FUNCTION_BLOCK PUBLIC SINT_TO_TestSuite EXTENDS TcUnit.FB_TestSuite
VAR
END_VAR

Check_SINT_TO_BOOL_Max();
Check_SINT_TO_BOOL_Min();
Check_SINT_TO_BYTE_Max();
Check_SINT_TO_BYTE_Min();
Check_SINT_TO_BYTE_TooLow();
Check_SINT_TO_WORD_Max();
Check_SINT_TO_WORD_Min();
Check_SINT_TO_WORD_TooLow();
Check_SINT_TO_DWORD_Max();
Check_SINT_TO_DWORD_Min();
Check_SINT_TO_DWORD_TooLow();
Check_SINT_TO_LWORD_Max();
Check_SINT_TO_LWORD_Min();
Check_SINT_TO_LWORD_TooLow();
Check_SINT_TO_SINT_Max();
Check_SINT_TO_SINT_Min();
Check_SINT_TO_INT_Max();
Check_SINT_TO_INT_Min();
Check_SINT_TO_DINT_Max();
Check_SINT_TO_DINT_Min();
Check_SINT_TO_LINT_Max();
Check_SINT_TO_LINT_Min();
Check_SINT_TO_USINT_Max();
Check_SINT_TO_USINT_Min();
Check_SINT_TO_USINT_TooLow();
Check_SINT_TO_UINT_Max();
Check_SINT_TO_UINT_Min();
Check_SINT_TO_UINT_TooLow();
Check_SINT_TO_UDINT_Max();
Check_SINT_TO_UDINT_Min();
Check_SINT_TO_UDINT_TooLow();
Check_SINT_TO_ULINT_Max();
Check_SINT_TO_ULINT_Min();
Check_SINT_TO_ULINT_TooLow();
Check_SINT_TO_REAL_Max();
Check_SINT_TO_REAL_Min();
Check_SINT_TO_LREAL_Max();
Check_SINT_TO_LREAL_Min();
Check_SINT_TO_TIME_Max();
Check_SINT_TO_TIME_Min();
Check_SINT_TO_TIME_TooLow();
Check_SINT_TO_TOD_Max();
Check_SINT_TO_TOD_Min();
Check_SINT_TO_TOD_TooLow();
Check_SINT_TO_DATE_Max();
Check_SINT_TO_DATE_Min();
Check_SINT_TO_DATE_TooLow();
Check_SINT_TO_DT_Max();
Check_SINT_TO_DT_Min();
Check_SINT_TO_DT_TooLow();
Check_SINT_TO_STRING_Max();
Check_SINT_TO_STRING_Min();

METHOD PUBLIC Check_SINT_TO_BOOL_Min
VAR
	value : SINT := DatatypeLimits.SINT_MIN_VALUE;
	actual : BOOL;
	converted : BOOL;
	equal : BOOL;
END_VAR
TEST('Check_SINT_TO_BOOL_Min');

// @TEST-RUN
converted := TryConvert_SINT_TO_Destination(value, actual);
equal := actual = SINT_TO_BOOL(value);

// @TEST-ASSERT
AssertTrue(Condition := equal, Message := 'Did not convert SINT to BOOL correctly');
AssertTrue(Condition := converted, Message := 'Did not report SINT to BOOL conversion was successful');

TEST_FINISHED();
END_METHOD

METHOD PUBLIC Check_SINT_TO_BOOL_Max
VAR
	value : SINT := DatatypeLimits.SINT_MAX_VALUE;
	actual : BOOL;
	converted : BOOL;
	equal : BOOL;
END_VAR
TEST('Check_SINT_TO_BOOL_Max');

// @TEST-RUN
converted := TryConvert_SINT_TO_Destination(value, actual);
equal := actual = SINT_TO_BOOL(value);

// @TEST-ASSERT
AssertTrue(Condition := equal, Message := 'Did not convert SINT to BOOL correctly');
AssertTrue(Condition := converted, Message := 'Did not report SINT to BOOL conversion was successful');

TEST_FINISHED();
END_METHOD

METHOD PUBLIC Check_SINT_TO_BYTE_Min
VAR
	value : SINT := DatatypeLimits.MIN_VALUE_OF_SINT_WHICH_CAN_BE_HELD_IN_A_BYTE;
	actual : BYTE;
	converted : BOOL;
	equal : BOOL;
END_VAR
TEST('Check_SINT_TO_BYTE_Min');

// @TEST-RUN
converted := TryConvert_SINT_TO_Destination(value, actual);
equal := actual = SINT_TO_BYTE(value);

// @TEST-ASSERT
AssertTrue(Condition := equal, Message := 'Did not convert SINT to BYTE correctly');
AssertTrue(Condition := converted, Message := 'Did not report SINT to BYTE conversion was successful');

TEST_FINISHED();
END_METHOD

METHOD PUBLIC Check_SINT_TO_BYTE_TooLow
VAR
	value : SINT := DatatypeLimits.SINT_MIN_VALUE;
	actual : BYTE;
	converted : BOOL;
END_VAR
TEST('Check_SINT_TO_BYTE_TooLow');

// @TEST-RUN
converted := TryConvert_SINT_TO_Destination(value, actual);

// @TEST-ASSERT
AssertFalse(Condition := converted, Message := 'Did not report SINT to BYTE conversion was prevented');

TEST_FINISHED();
END_METHOD

METHOD PUBLIC Check_SINT_TO_BYTE_Max
VAR
	value : SINT := DatatypeLimits.SINT_MAX_VALUE;
	actual : BYTE;
	converted : BOOL;
	equal : BOOL;
END_VAR
TEST('Check_SINT_TO_BYTE_Max');

// @TEST-RUN
converted := TryConvert_SINT_TO_Destination(value, actual);
equal := actual = SINT_TO_BYTE(value);

// @TEST-ASSERT
AssertTrue(Condition := equal, Message := 'Did not convert SINT to BYTE correctly');
AssertTrue(Condition := converted, Message := 'Did not report SINT to BYTE conversion was successful');

TEST_FINISHED();
END_METHOD

METHOD PUBLIC Check_SINT_TO_DATE_Min
VAR
	value : SINT := DatatypeLimits.MIN_VALUE_OF_SINT_WHICH_CAN_BE_HELD_IN_A_DATE;
	actual : DATE;
	converted : BOOL;
	equal : BOOL;
END_VAR
TEST('Check_SINT_TO_DATE_Min');

// @TEST-RUN
converted := TryConvert_SINT_TO_Destination(value, actual);
equal := actual = SINT_TO_DATE(value);

// @TEST-ASSERT
AssertTrue(Condition := equal, Message := 'Did not convert SINT to DATE correctly');
AssertTrue(Condition := converted, Message := 'Did not report SINT to DATE conversion was successful');

TEST_FINISHED();
END_METHOD

METHOD PUBLIC Check_SINT_TO_DATE_TooLow
VAR
	value : SINT := DatatypeLimits.SINT_MIN_VALUE;
	actual : DATE;
	converted : BOOL;
END_VAR
TEST('Check_SINT_TO_DATE_TooLow');

// @TEST-RUN
converted := TryConvert_SINT_TO_Destination(value, actual);

// @TEST-ASSERT
AssertFalse(Condition := converted, Message := 'Did not report SINT to DATE conversion was prevented');

TEST_FINISHED();
END_METHOD

METHOD PUBLIC Check_SINT_TO_DATE_Max
VAR
	value : SINT := DatatypeLimits.SINT_MAX_VALUE;
	actual : DATE;
	converted : BOOL;
	equal : BOOL;
END_VAR
TEST('Check_SINT_TO_DATE_Max');

// @TEST-RUN
converted := TryConvert_SINT_TO_Destination(value, actual);
equal := actual = SINT_TO_DATE(value);

// @TEST-ASSERT
AssertTrue(Condition := equal, Message := 'Did not convert SINT to DATE correctly');
AssertTrue(Condition := converted, Message := 'Did not report SINT to DATE conversion was successful');

TEST_FINISHED();
END_METHOD

METHOD PUBLIC Check_SINT_TO_DINT_Min
VAR
	value : SINT := DatatypeLimits.SINT_MIN_VALUE;
	actual : DINT;
	converted : BOOL;
	equal : BOOL;
END_VAR
TEST('Check_SINT_TO_DINT_Min');

// @TEST-RUN
converted := TryConvert_SINT_TO_Destination(value, actual);
equal := actual = SINT_TO_DINT(value);

// @TEST-ASSERT
AssertTrue(Condition := equal, Message := 'Did not convert SINT to DINT correctly');
AssertTrue(Condition := converted, Message := 'Did not report SINT to DINT conversion was successful');

TEST_FINISHED();
END_METHOD

METHOD PUBLIC Check_SINT_TO_DINT_Max
VAR
	value : SINT := DatatypeLimits.SINT_MAX_VALUE;
	actual : DINT;
	converted : BOOL;
	equal : BOOL;
END_VAR
TEST('Check_SINT_TO_DINT_Max');

// @TEST-RUN
converted := TryConvert_SINT_TO_Destination(value, actual);
equal := actual = SINT_TO_DINT(value);

// @TEST-ASSERT
AssertTrue(Condition := equal, Message := 'Did not convert SINT to DINT correctly');
AssertTrue(Condition := converted, Message := 'Did not report SINT to DINT conversion was successful');

TEST_FINISHED();
END_METHOD

METHOD PUBLIC Check_SINT_TO_DT_Min
VAR
	value : SINT := DatatypeLimits.MIN_VALUE_OF_SINT_WHICH_CAN_BE_HELD_IN_A_DT;
	actual : DT;
	converted : BOOL;
	equal : BOOL;
END_VAR
TEST('Check_SINT_TO_DT_Min');

// @TEST-RUN
converted := TryConvert_SINT_TO_Destination(value, actual);
equal := actual = SINT_TO_DT(value);

// @TEST-ASSERT
AssertTrue(Condition := equal, Message := 'Did not convert SINT to DT correctly');
AssertTrue(Condition := converted, Message := 'Did not report SINT to DT conversion was successful');

TEST_FINISHED();
END_METHOD

METHOD PUBLIC Check_SINT_TO_DT_TooLow
VAR
	value : SINT := DatatypeLimits.SINT_MIN_VALUE;
	actual : DT;
	converted : BOOL;
END_VAR
TEST('Check_SINT_TO_DT_TooLow');

// @TEST-RUN
converted := TryConvert_SINT_TO_Destination(value, actual);

// @TEST-ASSERT
AssertFalse(Condition := converted, Message := 'Did not report SINT to DT conversion was prevented');

TEST_FINISHED();
END_METHOD

METHOD PUBLIC Check_SINT_TO_DT_Max
VAR
	value : SINT := DatatypeLimits.SINT_MAX_VALUE;
	actual : DT;
	converted : BOOL;
	equal : BOOL;
END_VAR
TEST('Check_SINT_TO_DT_Max');

// @TEST-RUN
converted := TryConvert_SINT_TO_Destination(value, actual);
equal := actual = SINT_TO_DT(value);

// @TEST-ASSERT
AssertTrue(Condition := equal, Message := 'Did not convert SINT to DT correctly');
AssertTrue(Condition := converted, Message := 'Did not report SINT to DT conversion was successful');

TEST_FINISHED();
END_METHOD

METHOD PUBLIC Check_SINT_TO_DWORD_Min
VAR
	value : SINT := DatatypeLimits.MIN_VALUE_OF_SINT_WHICH_CAN_BE_HELD_IN_A_DWORD;
	actual : DWORD;
	converted : BOOL;
	equal : BOOL;
END_VAR
TEST('Check_SINT_TO_DWORD_Min');

// @TEST-RUN
converted := TryConvert_SINT_TO_Destination(value, actual);
equal := actual = SINT_TO_DWORD(value);

// @TEST-ASSERT
AssertTrue(Condition := equal, Message := 'Did not convert SINT to DWORD correctly');
AssertTrue(Condition := converted, Message := 'Did not report SINT to DWORD conversion was successful');

TEST_FINISHED();
END_METHOD

METHOD PUBLIC Check_SINT_TO_DWORD_TooLow
VAR
	value : SINT := DatatypeLimits.SINT_MIN_VALUE;
	actual : DWORD;
	converted : BOOL;
END_VAR
TEST('Check_SINT_TO_DWORD_TooLow');

// @TEST-RUN
converted := TryConvert_SINT_TO_Destination(value, actual);

// @TEST-ASSERT
AssertFalse(Condition := converted, Message := 'Did not report SINT to DWORD conversion was prevented');

TEST_FINISHED();
END_METHOD

METHOD PUBLIC Check_SINT_TO_DWORD_Max
VAR
	value : SINT := DatatypeLimits.SINT_MAX_VALUE;
	actual : DWORD;
	converted : BOOL;
	equal : BOOL;
END_VAR
TEST('Check_SINT_TO_DWORD_Max');

// @TEST-RUN
converted := TryConvert_SINT_TO_Destination(value, actual);
equal := actual = SINT_TO_DWORD(value);

// @TEST-ASSERT
AssertTrue(Condition := equal, Message := 'Did not convert SINT to DWORD correctly');
AssertTrue(Condition := converted, Message := 'Did not report SINT to DWORD conversion was successful');

TEST_FINISHED();
END_METHOD

METHOD PUBLIC Check_SINT_TO_INT_Min
VAR
	value : SINT := DatatypeLimits.SINT_MIN_VALUE;
	actual : INT;
	converted : BOOL;
	equal : BOOL;
END_VAR
TEST('Check_SINT_TO_INT_Min');

// @TEST-RUN
converted := TryConvert_SINT_TO_Destination(value, actual);
equal := actual = SINT_TO_INT(value);

// @TEST-ASSERT
AssertTrue(Condition := equal, Message := 'Did not convert SINT to INT correctly');
AssertTrue(Condition := converted, Message := 'Did not report SINT to INT conversion was successful');

TEST_FINISHED();
END_METHOD

METHOD PUBLIC Check_SINT_TO_INT_Max
VAR
	value : SINT := DatatypeLimits.SINT_MAX_VALUE;
	actual : INT;
	converted : BOOL;
	equal : BOOL;
END_VAR
TEST('Check_SINT_TO_INT_Max');

// @TEST-RUN
converted := TryConvert_SINT_TO_Destination(value, actual);
equal := actual = SINT_TO_INT(value);

// @TEST-ASSERT
AssertTrue(Condition := equal, Message := 'Did not convert SINT to INT correctly');
AssertTrue(Condition := converted, Message := 'Did not report SINT to INT conversion was successful');

TEST_FINISHED();
END_METHOD

METHOD PUBLIC Check_SINT_TO_LINT_Min
VAR
	value : SINT := DatatypeLimits.SINT_MIN_VALUE;
	actual : LINT;
	converted : BOOL;
	equal : BOOL;
END_VAR
TEST('Check_SINT_TO_LINT_Min');

// @TEST-RUN
converted := TryConvert_SINT_TO_Destination(value, actual);
equal := actual = SINT_TO_LINT(value);

// @TEST-ASSERT
AssertTrue(Condition := equal, Message := 'Did not convert SINT to LINT correctly');
AssertTrue(Condition := converted, Message := 'Did not report SINT to LINT conversion was successful');

TEST_FINISHED();
END_METHOD

METHOD PUBLIC Check_SINT_TO_LINT_Max
VAR
	value : SINT := DatatypeLimits.SINT_MAX_VALUE;
	actual : LINT;
	converted : BOOL;
	equal : BOOL;
END_VAR
TEST('Check_SINT_TO_LINT_Max');

// @TEST-RUN
converted := TryConvert_SINT_TO_Destination(value, actual);
equal := actual = SINT_TO_LINT(value);

// @TEST-ASSERT
AssertTrue(Condition := equal, Message := 'Did not convert SINT to LINT correctly');
AssertTrue(Condition := converted, Message := 'Did not report SINT to LINT conversion was successful');

TEST_FINISHED();
END_METHOD

METHOD PUBLIC Check_SINT_TO_LREAL_Min
VAR
	value : SINT := DatatypeLimits.SINT_MIN_VALUE;
	actual : LREAL;
	converted : BOOL;
	equal : BOOL;
END_VAR
TEST('Check_SINT_TO_LREAL_Min');

// @TEST-RUN
converted := TryConvert_SINT_TO_Destination(value, actual);
equal := actual = SINT_TO_LREAL(value);

// @TEST-ASSERT
AssertTrue(Condition := equal, Message := 'Did not convert SINT to LREAL correctly');
AssertTrue(Condition := converted, Message := 'Did not report SINT to LREAL conversion was successful');

TEST_FINISHED();
END_METHOD

METHOD PUBLIC Check_SINT_TO_LREAL_Max
VAR
	value : SINT := DatatypeLimits.SINT_MAX_VALUE;
	actual : LREAL;
	converted : BOOL;
	equal : BOOL;
END_VAR
TEST('Check_SINT_TO_LREAL_Max');

// @TEST-RUN
converted := TryConvert_SINT_TO_Destination(value, actual);
equal := actual = SINT_TO_LREAL(value);

// @TEST-ASSERT
AssertTrue(Condition := equal, Message := 'Did not convert SINT to LREAL correctly');
AssertTrue(Condition := converted, Message := 'Did not report SINT to LREAL conversion was successful');

TEST_FINISHED();
END_METHOD

METHOD PUBLIC Check_SINT_TO_LWORD_Min
VAR
	value : SINT := DatatypeLimits.MIN_VALUE_OF_SINT_WHICH_CAN_BE_HELD_IN_A_LWORD;
	actual : LWORD;
	converted : BOOL;
	equal : BOOL;
END_VAR
TEST('Check_SINT_TO_LWORD_Min');

// @TEST-RUN
converted := TryConvert_SINT_TO_Destination(value, actual);
equal := actual = SINT_TO_LWORD(value);

// @TEST-ASSERT
AssertTrue(Condition := equal, Message := 'Did not convert SINT to LWORD correctly');
AssertTrue(Condition := converted, Message := 'Did not report SINT to LWORD conversion was successful');

TEST_FINISHED();
END_METHOD

METHOD PUBLIC Check_SINT_TO_LWORD_TooLow
VAR
	value : SINT := DatatypeLimits.SINT_MIN_VALUE;
	actual : LWORD;
	converted : BOOL;
END_VAR
TEST('Check_SINT_TO_LWORD_TooLow');

// @TEST-RUN
converted := TryConvert_SINT_TO_Destination(value, actual);

// @TEST-ASSERT
AssertFalse(Condition := converted, Message := 'Did not report SINT to LWORD conversion was prevented');

TEST_FINISHED();
END_METHOD

METHOD PUBLIC Check_SINT_TO_LWORD_Max
VAR
	value : SINT := DatatypeLimits.SINT_MAX_VALUE;
	actual : LWORD;
	converted : BOOL;
	equal : BOOL;
END_VAR
TEST('Check_SINT_TO_LWORD_Max');

// @TEST-RUN
converted := TryConvert_SINT_TO_Destination(value, actual);
equal := actual = SINT_TO_LWORD(value);

// @TEST-ASSERT
AssertTrue(Condition := equal, Message := 'Did not convert SINT to LWORD correctly');
AssertTrue(Condition := converted, Message := 'Did not report SINT to LWORD conversion was successful');

TEST_FINISHED();
END_METHOD

METHOD PUBLIC Check_SINT_TO_REAL_Min
VAR
	value : SINT := DatatypeLimits.SINT_MIN_VALUE;
	actual : REAL;
	converted : BOOL;
	equal : BOOL;
END_VAR
TEST('Check_SINT_TO_REAL_Min');

// @TEST-RUN
converted := TryConvert_SINT_TO_Destination(value, actual);
equal := actual = SINT_TO_REAL(value);

// @TEST-ASSERT
AssertTrue(Condition := equal, Message := 'Did not convert SINT to REAL correctly');
AssertTrue(Condition := converted, Message := 'Did not report SINT to REAL conversion was successful');

TEST_FINISHED();
END_METHOD

METHOD PUBLIC Check_SINT_TO_REAL_Max
VAR
	value : SINT := DatatypeLimits.SINT_MAX_VALUE;
	actual : REAL;
	converted : BOOL;
	equal : BOOL;
END_VAR
TEST('Check_SINT_TO_REAL_Max');

// @TEST-RUN
converted := TryConvert_SINT_TO_Destination(value, actual);
equal := actual = SINT_TO_REAL(value);

// @TEST-ASSERT
AssertTrue(Condition := equal, Message := 'Did not convert SINT to REAL correctly');
AssertTrue(Condition := converted, Message := 'Did not report SINT to REAL conversion was successful');

TEST_FINISHED();
END_METHOD

METHOD PUBLIC Check_SINT_TO_SINT_Min
VAR
	value : SINT := DatatypeLimits.SINT_MIN_VALUE;
	actual : SINT;
	converted : BOOL;
	equal : BOOL;
END_VAR
TEST('Check_SINT_TO_SINT_Min');

// @TEST-RUN
converted := TryConvert_SINT_TO_Destination(value, actual);
equal := actual = value;

// @TEST-ASSERT
AssertTrue(Condition := equal, Message := 'Did not convert SINT to SINT correctly');
AssertTrue(Condition := converted, Message := 'Did not report SINT to SINT conversion was successful');

TEST_FINISHED();
END_METHOD

METHOD PUBLIC Check_SINT_TO_SINT_Max
VAR
	value : SINT := DatatypeLimits.SINT_MAX_VALUE;
	actual : SINT;
	converted : BOOL;
	equal : BOOL;
END_VAR
TEST('Check_SINT_TO_SINT_Max');

// @TEST-RUN
converted := TryConvert_SINT_TO_Destination(value, actual);
equal := actual = value;

// @TEST-ASSERT
AssertTrue(Condition := equal, Message := 'Did not convert SINT to SINT correctly');
AssertTrue(Condition := converted, Message := 'Did not report SINT to SINT conversion was successful');

TEST_FINISHED();
END_METHOD

METHOD PUBLIC Check_SINT_TO_STRING_Min
VAR
	value : SINT := DatatypeLimits.SINT_MIN_VALUE;
	actual : STRING;
	converted : BOOL;
	equal : BOOL;
END_VAR
TEST('Check_SINT_TO_STRING_Min');

// @TEST-RUN
converted := TryConvert_SINT_TO_Destination(value, actual);
equal := actual = SINT_TO_STRING(value);

// @TEST-ASSERT
AssertTrue(Condition := equal, Message := 'Did not convert SINT to STRING correctly');
AssertTrue(Condition := converted, Message := 'Did not report SINT to STRING conversion was successful');

TEST_FINISHED();
END_METHOD

METHOD PUBLIC Check_SINT_TO_STRING_Max
VAR
	value : SINT := DatatypeLimits.SINT_MAX_VALUE;
	actual : STRING;
	converted : BOOL;
	equal : BOOL;
END_VAR
TEST('Check_SINT_TO_STRING_Max');

// @TEST-RUN
converted := TryConvert_SINT_TO_Destination(value, actual);
equal := actual = SINT_TO_STRING(value);

// @TEST-ASSERT
AssertTrue(Condition := equal, Message := 'Did not convert SINT to STRING correctly');
AssertTrue(Condition := converted, Message := 'Did not report SINT to STRING conversion was successful');

TEST_FINISHED();
END_METHOD

METHOD PUBLIC Check_SINT_TO_TIME_Min
VAR
	value : SINT := DatatypeLimits.MIN_VALUE_OF_SINT_WHICH_CAN_BE_HELD_IN_A_TIME;
	actual : TIME;
	converted : BOOL;
	equal : BOOL;
END_VAR
TEST('Check_SINT_TO_TIME_Min');

// @TEST-RUN
converted := TryConvert_SINT_TO_Destination(value, actual);
equal := actual = SINT_TO_TIME(value);

// @TEST-ASSERT
AssertTrue(Condition := equal, Message := 'Did not convert SINT to TIME correctly');
AssertTrue(Condition := converted, Message := 'Did not report SINT to TIME conversion was successful');

TEST_FINISHED();
END_METHOD

METHOD PUBLIC Check_SINT_TO_TIME_TooLow
VAR
	value : SINT := DatatypeLimits.SINT_MIN_VALUE;
	actual : TIME;
	converted : BOOL;
END_VAR
TEST('Check_SINT_TO_TIME_TooLow');

// @TEST-RUN
converted := TryConvert_SINT_TO_Destination(value, actual);

// @TEST-ASSERT
AssertFalse(Condition := converted, Message := 'Did not report SINT to TIME conversion was prevented');

TEST_FINISHED();
END_METHOD

METHOD PUBLIC Check_SINT_TO_TIME_Max
VAR
	value : SINT := DatatypeLimits.SINT_MAX_VALUE;
	actual : TIME;
	converted : BOOL;
	equal : BOOL;
END_VAR
TEST('Check_SINT_TO_TIME_Max');

// @TEST-RUN
converted := TryConvert_SINT_TO_Destination(value, actual);
equal := actual = SINT_TO_TIME(value);

// @TEST-ASSERT
AssertTrue(Condition := equal, Message := 'Did not convert SINT to TIME correctly');
AssertTrue(Condition := converted, Message := 'Did not report SINT to TIME conversion was successful');

TEST_FINISHED();
END_METHOD

METHOD PUBLIC Check_SINT_TO_TOD_Min
VAR
	value : SINT := DatatypeLimits.MIN_VALUE_OF_SINT_WHICH_CAN_BE_HELD_IN_A_TOD;
	actual : TOD;
	converted : BOOL;
	equal : BOOL;
END_VAR
TEST('Check_SINT_TO_TOD_Min');

// @TEST-RUN
converted := TryConvert_SINT_TO_Destination(value, actual);
equal := actual = SINT_TO_TOD(value);

// @TEST-ASSERT
AssertTrue(Condition := equal, Message := 'Did not convert SINT to TOD correctly');
AssertTrue(Condition := converted, Message := 'Did not report SINT to TOD conversion was successful');

TEST_FINISHED();
END_METHOD

METHOD PUBLIC Check_SINT_TO_TOD_TooLow
VAR
	value : SINT := DatatypeLimits.SINT_MIN_VALUE;
	actual : TOD;
	converted : BOOL;
END_VAR
TEST('Check_SINT_TO_TOD_TooLow');

// @TEST-RUN
converted := TryConvert_SINT_TO_Destination(value, actual);

// @TEST-ASSERT
AssertFalse(Condition := converted, Message := 'Did not report SINT to TOD conversion was prevented');

TEST_FINISHED();
END_METHOD

METHOD PUBLIC Check_SINT_TO_TOD_Max
VAR
	value : SINT := DatatypeLimits.SINT_MAX_VALUE;
	actual : TOD;
	converted : BOOL;
	equal : BOOL;
END_VAR
TEST('Check_SINT_TO_TOD_Max');

// @TEST-RUN
converted := TryConvert_SINT_TO_Destination(value, actual);
equal := actual = SINT_TO_TOD(value);

// @TEST-ASSERT
AssertTrue(Condition := equal, Message := 'Did not convert SINT to TOD correctly');
AssertTrue(Condition := converted, Message := 'Did not report SINT to TOD conversion was successful');

TEST_FINISHED();
END_METHOD

METHOD PUBLIC Check_SINT_TO_UDINT_Min
VAR
	value : SINT := DatatypeLimits.MIN_VALUE_OF_SINT_WHICH_CAN_BE_HELD_IN_A_UDINT;
	actual : UDINT;
	converted : BOOL;
	equal : BOOL;
END_VAR
TEST('Check_SINT_TO_UDINT_Min');

// @TEST-RUN
converted := TryConvert_SINT_TO_Destination(value, actual);
equal := actual = SINT_TO_UDINT(value);

// @TEST-ASSERT
AssertTrue(Condition := equal, Message := 'Did not convert SINT to UDINT correctly');
AssertTrue(Condition := converted, Message := 'Did not report SINT to UDINT conversion was successful');

TEST_FINISHED();
END_METHOD

METHOD PUBLIC Check_SINT_TO_UDINT_TooLow
VAR
	value : SINT := DatatypeLimits.SINT_MIN_VALUE;
	actual : UDINT;
	converted : BOOL;
END_VAR
TEST('Check_SINT_TO_UDINT_TooLow');

// @TEST-RUN
converted := TryConvert_SINT_TO_Destination(value, actual);

// @TEST-ASSERT
AssertFalse(Condition := converted, Message := 'Did not report SINT to UDINT conversion was prevented');

TEST_FINISHED();
END_METHOD

METHOD PUBLIC Check_SINT_TO_UDINT_Max
VAR
	value : SINT := DatatypeLimits.SINT_MAX_VALUE;
	actual : UDINT;
	converted : BOOL;
	equal : BOOL;
END_VAR
TEST('Check_SINT_TO_UDINT_Max');

// @TEST-RUN
converted := TryConvert_SINT_TO_Destination(value, actual);
equal := actual = SINT_TO_UDINT(value);

// @TEST-ASSERT
AssertTrue(Condition := equal, Message := 'Did not convert SINT to UDINT correctly');
AssertTrue(Condition := converted, Message := 'Did not report SINT to UDINT conversion was successful');

TEST_FINISHED();
END_METHOD

METHOD PUBLIC Check_SINT_TO_UINT_Min
VAR
	value : SINT := DatatypeLimits.MIN_VALUE_OF_SINT_WHICH_CAN_BE_HELD_IN_A_UINT;
	actual : UINT;
	converted : BOOL;
	equal : BOOL;
END_VAR
TEST('Check_SINT_TO_UINT_Min');

// @TEST-RUN
converted := TryConvert_SINT_TO_Destination(value, actual);
equal := actual = SINT_TO_UINT(value);

// @TEST-ASSERT
AssertTrue(Condition := equal, Message := 'Did not convert SINT to UINT correctly');
AssertTrue(Condition := converted, Message := 'Did not report SINT to UINT conversion was successful');

TEST_FINISHED();
END_METHOD

METHOD PUBLIC Check_SINT_TO_UINT_TooLow
VAR
	value : SINT := DatatypeLimits.SINT_MIN_VALUE;
	actual : UINT;
	converted : BOOL;
END_VAR
TEST('Check_SINT_TO_UINT_TooLow');

// @TEST-RUN
converted := TryConvert_SINT_TO_Destination(value, actual);

// @TEST-ASSERT
AssertFalse(Condition := converted, Message := 'Did not report SINT to UINT conversion was prevented');

TEST_FINISHED();
END_METHOD

METHOD PUBLIC Check_SINT_TO_UINT_Max
VAR
	value : SINT := DatatypeLimits.SINT_MAX_VALUE;
	actual : UINT;
	converted : BOOL;
	equal : BOOL;
END_VAR
TEST('Check_SINT_TO_UINT_Max');

// @TEST-RUN
converted := TryConvert_SINT_TO_Destination(value, actual);
equal := actual = SINT_TO_UINT(value);

// @TEST-ASSERT
AssertTrue(Condition := equal, Message := 'Did not convert SINT to UINT correctly');
AssertTrue(Condition := converted, Message := 'Did not report SINT to UINT conversion was successful');

TEST_FINISHED();
END_METHOD

METHOD PUBLIC Check_SINT_TO_ULINT_Min
VAR
	value : SINT := DatatypeLimits.MIN_VALUE_OF_SINT_WHICH_CAN_BE_HELD_IN_A_ULINT;
	actual : ULINT;
	converted : BOOL;
	equal : BOOL;
END_VAR
TEST('Check_SINT_TO_ULINT_Min');

// @TEST-RUN
converted := TryConvert_SINT_TO_Destination(value, actual);
equal := actual = SINT_TO_ULINT(value);

// @TEST-ASSERT
AssertTrue(Condition := equal, Message := 'Did not convert SINT to ULINT correctly');
AssertTrue(Condition := converted, Message := 'Did not report SINT to ULINT conversion was successful');

TEST_FINISHED();
END_METHOD

METHOD PUBLIC Check_SINT_TO_ULINT_TooLow
VAR
	value : SINT := DatatypeLimits.SINT_MIN_VALUE;
	actual : ULINT;
	converted : BOOL;
END_VAR
TEST('Check_SINT_TO_ULINT_TooLow');

// @TEST-RUN
converted := TryConvert_SINT_TO_Destination(value, actual);

// @TEST-ASSERT
AssertFalse(Condition := converted, Message := 'Did not report SINT to ULINT conversion was prevented');

TEST_FINISHED();
END_METHOD

METHOD PUBLIC Check_SINT_TO_ULINT_Max
VAR
	value : SINT := DatatypeLimits.SINT_MAX_VALUE;
	actual : ULINT;
	converted : BOOL;
	equal : BOOL;
END_VAR
TEST('Check_SINT_TO_ULINT_Max');

// @TEST-RUN
converted := TryConvert_SINT_TO_Destination(value, actual);
equal := actual = SINT_TO_ULINT(value);

// @TEST-ASSERT
AssertTrue(Condition := equal, Message := 'Did not convert SINT to ULINT correctly');
AssertTrue(Condition := converted, Message := 'Did not report SINT to ULINT conversion was successful');

TEST_FINISHED();
END_METHOD

METHOD PUBLIC Check_SINT_TO_USINT_Min
VAR
	value : SINT := DatatypeLimits.MIN_VALUE_OF_SINT_WHICH_CAN_BE_HELD_IN_A_USINT;
	actual : USINT;
	converted : BOOL;
	equal : BOOL;
END_VAR
TEST('Check_SINT_TO_USINT_Min');

// @TEST-RUN
converted := TryConvert_SINT_TO_Destination(value, actual);
equal := actual = SINT_TO_USINT(value);

// @TEST-ASSERT
AssertTrue(Condition := equal, Message := 'Did not convert SINT to USINT correctly');
AssertTrue(Condition := converted, Message := 'Did not report SINT to USINT conversion was successful');

TEST_FINISHED();
END_METHOD

METHOD PUBLIC Check_SINT_TO_USINT_TooLow
VAR
	value : SINT := DatatypeLimits.SINT_MIN_VALUE;
	actual : USINT;
	converted : BOOL;
END_VAR
TEST('Check_SINT_TO_USINT_TooLow');

// @TEST-RUN
converted := TryConvert_SINT_TO_Destination(value, actual);

// @TEST-ASSERT
AssertFalse(Condition := converted, Message := 'Did not report SINT to USINT conversion was prevented');

TEST_FINISHED();
END_METHOD

METHOD PUBLIC Check_SINT_TO_USINT_Max
VAR
	value : SINT := DatatypeLimits.SINT_MAX_VALUE;
	actual : USINT;
	converted : BOOL;
	equal : BOOL;
END_VAR
TEST('Check_SINT_TO_USINT_Max');

// @TEST-RUN
converted := TryConvert_SINT_TO_Destination(value, actual);
equal := actual = SINT_TO_USINT(value);

// @TEST-ASSERT
AssertTrue(Condition := equal, Message := 'Did not convert SINT to USINT correctly');
AssertTrue(Condition := converted, Message := 'Did not report SINT to USINT conversion was successful');

TEST_FINISHED();
END_METHOD

METHOD PUBLIC Check_SINT_TO_WORD_Min
VAR
	value : SINT := DatatypeLimits.MIN_VALUE_OF_SINT_WHICH_CAN_BE_HELD_IN_A_WORD;
	actual : WORD;
	converted : BOOL;
	equal : BOOL;
END_VAR
TEST('Check_SINT_TO_WORD_Min');

// @TEST-RUN
converted := TryConvert_SINT_TO_Destination(value, actual);
equal := actual = SINT_TO_WORD(value);

// @TEST-ASSERT
AssertTrue(Condition := equal, Message := 'Did not convert SINT to WORD correctly');
AssertTrue(Condition := converted, Message := 'Did not report SINT to WORD conversion was successful');

TEST_FINISHED();
END_METHOD

METHOD PUBLIC Check_SINT_TO_WORD_TooLow
VAR
	value : SINT := DatatypeLimits.SINT_MIN_VALUE;
	actual : WORD;
	converted : BOOL;
END_VAR
TEST('Check_SINT_TO_WORD_TooLow');

// @TEST-RUN
converted := TryConvert_SINT_TO_Destination(value, actual);

// @TEST-ASSERT
AssertFalse(Condition := converted, Message := 'Did not report SINT to WORD conversion was prevented');

TEST_FINISHED();
END_METHOD

METHOD PUBLIC Check_SINT_TO_WORD_Max
VAR
	value : SINT := DatatypeLimits.SINT_MAX_VALUE;
	actual : WORD;
	converted : BOOL;
	equal : BOOL;
END_VAR
TEST('Check_SINT_TO_WORD_Max');

// @TEST-RUN
converted := TryConvert_SINT_TO_Destination(value, actual);
equal := actual = SINT_TO_WORD(value);

// @TEST-ASSERT
AssertTrue(Condition := equal, Message := 'Did not convert SINT to WORD correctly');
AssertTrue(Condition := converted, Message := 'Did not report SINT to WORD conversion was successful');

TEST_FINISHED();
END_METHOD

END_FUNCTION_BLOCK

(* stored: Version 1.1.0.1, ProductVersion 3.1.4024.12
   POU SINT_TO_TestSuite: Id {d2935109-592a-4660-a8c8-4060d6714044}, SpecialFunc None
   Method Check_SINT_TO_BOOL_Min: Id {b4e1f5ea-a868-42a5-badf-1c2fe6e474bf}
   Method Check_SINT_TO_BOOL_Max: Id {6a2e4cb8-bd22-40da-a63c-023c440de75b}
   Method Check_SINT_TO_BYTE_Min: Id {f33d30b4-fb45-4db5-b495-92d8c1be4e0d}
   Method Check_SINT_TO_BYTE_TooLow: Id {8da1fcb5-2a9e-4304-921b-105444f4a9da}
   Method Check_SINT_TO_BYTE_Max: Id {b7af06c5-ef60-4ce5-a614-3cf717914206}
   Method Check_SINT_TO_DATE_Min: Id {bf03900b-05b9-4b28-87e2-be08ff069d64}
   Method Check_SINT_TO_DATE_TooLow: Id {00895fa3-c1d3-4036-a103-755a25149ebb}
   Method Check_SINT_TO_DATE_Max: Id {d91b2e4f-15e3-43c3-bf64-989c31456b0b}
   Method Check_SINT_TO_DINT_Min: Id {40f42476-e11e-4c5c-b29b-1d625aeb0e28}
   Method Check_SINT_TO_DINT_Max: Id {6cb791d0-d5db-4d0d-ad4e-25eb7167f62a}
   Method Check_SINT_TO_DT_Min: Id {ba3605d1-4ae1-49a8-913f-f05511458d02}
   Method Check_SINT_TO_DT_TooLow: Id {df9b3847-bd7f-4d8f-b337-f908d2e1c66c}
   Method Check_SINT_TO_DT_Max: Id {71f25761-6888-4de3-9dc6-22de9e170abf}
   Method Check_SINT_TO_DWORD_Min: Id {3e387a88-401d-4221-91b5-281691f40c04}
   Method Check_SINT_TO_DWORD_TooLow: Id {6bcc7820-a37c-40f1-bcfb-796df12e614a}
   Method Check_SINT_TO_DWORD_Max: Id {3c54819b-072a-4563-917f-92f1de18d882}
   Method Check_SINT_TO_INT_Min: Id {8fbec2a1-d2c2-4853-99a8-d24ca453e639}
   Method Check_SINT_TO_INT_Max: Id {9216db9d-9329-4bf5-90ce-569042c61e5e}
   Method Check_SINT_TO_LINT_Min: Id {14d81d3a-1ee6-455e-8948-c185937a2ab0}
   Method Check_SINT_TO_LINT_Max: Id {593f90c6-8e09-4e49-be21-5a716064a765}
   Method Check_SINT_TO_LREAL_Min: Id {b489d038-ea5b-4915-8886-cf2784d003dc}
   Method Check_SINT_TO_LREAL_Max: Id {ee483dc3-9ae9-441b-a030-e0a5642fe5dd}
   Method Check_SINT_TO_LWORD_Min: Id {d43962e1-ab2d-4a6e-b4af-5ef07cc726bd}
   Method Check_SINT_TO_LWORD_TooLow: Id {9f717789-6210-40d8-9c75-fc289d6ab3e7}
   Method Check_SINT_TO_LWORD_Max: Id {69369c34-2e90-4bbd-8d2c-23f6d4be26b5}
   Method Check_SINT_TO_REAL_Min: Id {7d5d602a-b046-4251-a378-cb71a2be4230}
   Method Check_SINT_TO_REAL_Max: Id {4c6368af-1cbb-4072-9d05-5a70e4717849}
   Method Check_SINT_TO_SINT_Min: Id {aefbfa88-1176-4666-af3c-5ce1ce644a85}
   Method Check_SINT_TO_SINT_Max: Id {b164d6eb-9ef3-404f-847d-11bc774c89d1}
   Method Check_SINT_TO_STRING_Min: Id {f8a77fae-20fa-470f-8898-2c6d67152324}
   Method Check_SINT_TO_STRING_Max: Id {c4d4c69f-d3ab-40c3-bff1-c1e8915ed708}
   Method Check_SINT_TO_TIME_Min: Id {d3ab607e-5948-41b8-9459-e3e871cfec53}
   Method Check_SINT_TO_TIME_TooLow: Id {6937bed0-0311-479d-a41e-fa1ac5d6f7a5}
   Method Check_SINT_TO_TIME_Max: Id {6f11779f-31ec-479f-b446-90acdd7db6a0}
   Method Check_SINT_TO_TOD_Min: Id {14fae61c-b47f-48c1-bbc5-4ebd8ed62f71}
   Method Check_SINT_TO_TOD_TooLow: Id {3b9d679f-5257-4a0a-9338-88395a27906f}
   Method Check_SINT_TO_TOD_Max: Id {787c4e9e-b5f1-4366-bbe0-2d965143225a}
   Method Check_SINT_TO_UDINT_Min: Id {84ebcaed-29cf-48cd-af68-368c9ed4d701}
   Method Check_SINT_TO_UDINT_TooLow: Id {20cdfb93-4116-482f-a768-8554d7cb23b4}
   Method Check_SINT_TO_UDINT_Max: Id {bb39e633-0de4-4f90-b3c4-24b857185546}
   Method Check_SINT_TO_UINT_Min: Id {ea4bf66e-49ab-42a4-9a13-9c9bd843bdc0}
   Method Check_SINT_TO_UINT_TooLow: Id {ed773e2e-523b-4467-8361-e8f66b20df3c}
   Method Check_SINT_TO_UINT_Max: Id {6bda5c26-036a-4914-9c9c-8404caa0c3da}
   Method Check_SINT_TO_ULINT_Min: Id {b65951e6-2025-4884-bb03-8d80d08e246b}
   Method Check_SINT_TO_ULINT_TooLow: Id {bf872a84-92f2-4e5b-9442-78b792781aa1}
   Method Check_SINT_TO_ULINT_Max: Id {471bd500-a610-45fb-ba86-721dcee6da88}
   Method Check_SINT_TO_USINT_Min: Id {1f417970-bd87-40be-a947-673b6cbe0353}
   Method Check_SINT_TO_USINT_TooLow: Id {a11cc494-78c6-4b3e-bde7-112a428fb65c}
   Method Check_SINT_TO_USINT_Max: Id {868eeff5-bf77-4df4-b805-6838eb5affca}
   Method Check_SINT_TO_WORD_Min: Id {1bbf01a8-c443-40e9-85e4-61883f7b38cb}
   Method Check_SINT_TO_WORD_TooLow: Id {e140dada-602d-44c0-b950-9b3bb6244ac4}
   Method Check_SINT_TO_WORD_Max: Id {d80fc6dc-aeea-4280-90a1-b58a8e89c164} *)
